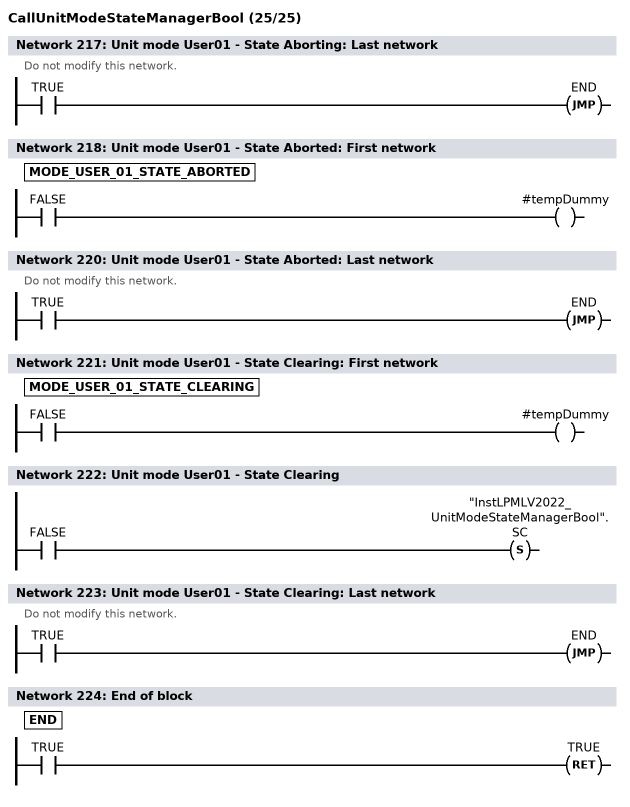
   RUNG wire#powerrail
      Contact( TRUE )
      JumpCoil( END )
   END_RUNG
   // the same network as SCL:
   IF TRUE THEN GOTO END; END_IF;
END_REGION

REGION Network 218: Unit mode User01 - State Aborted: First network
   Label( MODE_USER_01_STATE_ABORTED )
   RUNG wire#powerrail
      Contact( FALSE )
      Coil( #tempDummy )
   END_RUNG
   // the same network as SCL:
   MODE_USER_01_STATE_ABORTED:
   #tempDummy := FALSE;
END_REGION

REGION Network 219: Unit mode User01 - State Aborted
END_REGION

REGION Network 220: Unit mode User01 - State Aborted: Last network
   // Do not modify this network.
   RUNG wire#powerrail
      Contact( TRUE )
      JumpCoil( END )
   END_RUNG
   // the same network as SCL:
   IF TRUE THEN GOTO END; END_IF;
END_REGION

REGION Network 221: Unit mode User01 - State Clearing: First network
   Label( MODE_USER_01_STATE_CLEARING )
   RUNG wire#powerrail
      Contact( FALSE )
      Coil( #tempDummy )
   END_RUNG
   // the same network as SCL:
   MODE_USER_01_STATE_CLEARING:
   #tempDummy := FALSE;
END_REGION

REGION Network 222: Unit mode User01 - State Clearing
   RUNG wire#powerrail
      Contact( FALSE )
      S_Coil( "InstLPMLV2022_UnitModeStateManagerBool".SC )
   END_RUNG
   // the same network as SCL:
   IF FALSE THEN "InstLPMLV2022_UnitModeStateManagerBool".SC := TRUE; END_IF;
END_REGION

REGION Network 223: Unit mode User01 - State Clearing: Last network
   // Do not modify this network.
   RUNG wire#powerrail
      Contact( TRUE )
      JumpCoil( END )
   END_RUNG
   // the same network as SCL:
   IF TRUE THEN GOTO END; END_IF;
END_REGION

REGION Network 224: End of block
   Label( END )
   RUNG wire#powerrail
      Contact( TRUE )
      ReturnCoil( TRUE )
   END_RUNG
   // the same network as SCL:
   END:
   IF TRUE THEN
       ENO := TRUE;
       RETURN;
   END_IF;
END_REGION
END_FUNCTION_BLOCK
